{attribute addProperty BoxType "EK1122-0000-0018"}
{attribute addProperty Id "Beckhoff_EPP9xxxsub_EK1100EK1100_179A0949162A_0001_EPP9001_0060_0016EPP9001_179A0949162A_0002_EPP9001_0060_0017EPP9001_179A0949162A_0003_EPP9022_0060_0017EPP9022_497E3BE925632A_0004_EPP9022_9060_0017EPP9022_497E3BE925632"}
{attribute addProperty CRC "1883167374"}
{attribute addProperty SizeInBites "560"}
{attribute addProperty SizeInBytes "70"}
TYPE Beckhoff_EPP9xxxEK1122_703EDA8E EXTENDS EK1122_179A0949 :
STRUCT
	{attribute addProperty Name "Beckhoff_EPP9xxxsub_EK1100"}
	Beckhoff_EPP9xxxsub_EK1100 : EK1100_179A0949;
	{attribute addProperty Name "A_0001_EPP9001_0060_0016"}
	A_0001_EPP9001_0060_0016 : EPP9001_179A0949;
	{attribute addProperty Name "A_0002_EPP9001_0060_0017"}
	A_0002_EPP9001_0060_0017 : EPP9001_179A0949;
	{attribute addProperty Name "A_0003_EPP9022_0060_0017"}
	A_0003_EPP9022_0060_0017 : EPP9022_497E3BE9;
	{attribute addProperty Name "A_0004_EPP9022_9060_0017"}
	A_0004_EPP9022_9060_0017 : EPP9022_497E3BE9;
END_STRUCT
END_TYPE

(* stored: Version 1.2.0.0, ProductVersion 3.1.4024.9
   DUT Beckhoff_EPP9xxxEK1122_703EDA8E: Id {9b819845-e3f9-458f-bef6-ede13eab5c59} *)
